// TIA Portal project "tezTia" (V14)

(* hardware
DEVICE "S7-1200 station_1"  S7-1200 Station
   slot 0: "Rack_0"  Rack  V1.0
   slot 1: "PLC_1"  CPU 1215C AC/DC/Rly  6ES7 215-1BG31-0XB0  V3.0
*)

// ===== PLC "PLC_1"  CPU 1215C AC/DC/Rly =====

VAR_GLOBAL   // PLC tag table "Default tag table"
   "start" AT %I0.0 : Bool;
   "stop" AT %I0.1 : Bool;
   "renk sensörü" AT %IW64 : Word;
   "kamera" AT %QW80 : Word;
   "motor" AT %Q0.0 : Bool;
   "motor_1" AT %Q0.1 : Bool;
   "motor_2" AT %Q0.2 : Bool;
   "motor_3" AT %Q0.3 : Bool;
   "motor_4" AT %Q0.4 : Bool;
   "kırmızı" AT %M40.0 : Bool;
   "yeşil" AT %M40.1 : Bool;
   "mavi" AT %M40.2 : Bool;
   "bozuk" AT %M40.3 : Bool;
   "motor_3 geri" AT %Q0.6 : Bool;
END_VAR

DATA_BLOCK "çark çevir_DB"   // DB6
{ S7_Optimized_Access := 'TRUE' }
VERSION : 0.1
// stored: InstanceOfName çark çevir
"çark çevir"
BEGIN
END_DATA_BLOCK

DATA_BLOCK "şekil algıla_DB"   // DB7
{ S7_Optimized_Access := 'TRUE' }
VERSION : 0.1
// stored: InstanceOfName şekil algıla
"şekil algıla"
BEGIN
END_DATA_BLOCK

DATA_BLOCK "reset_DB"   // DB9
{ S7_Optimized_Access := 'TRUE' }
VERSION : 0.1
// stored: InstanceOfName reset
"reset"
BEGIN
END_DATA_BLOCK

// folder: System blocks/Program resources

DATA_BLOCK "IEC_Timer_0_DB"   // DB1
{ S7_Optimized_Access := 'TRUE' }
AUTHOR : Simatic
FAMILY : IEC
NAME : IEC_TMR
VERSION : 1.0
// stored: InstanceOfName IEC_TIMER
"IEC_TIMER"
BEGIN
END_DATA_BLOCK

DATA_BLOCK "IEC_Timer_0_DB_1"   // DB2
{ S7_Optimized_Access := 'TRUE' }
AUTHOR : Simatic
FAMILY : IEC
NAME : IEC_TMR
VERSION : 1.0
// stored: InstanceOfName IEC_TIMER
"IEC_TIMER"
BEGIN
END_DATA_BLOCK

DATA_BLOCK "IEC_Timer_0_DB_2"   // DB3
{ S7_Optimized_Access := 'TRUE' }
AUTHOR : Simatic
FAMILY : IEC
NAME : IEC_TMR
VERSION : 1.0
// stored: InstanceOfName IEC_TIMER
"IEC_TIMER"
BEGIN
END_DATA_BLOCK

DATA_BLOCK "IEC_Timer_0_DB_3"   // DB4
{ S7_Optimized_Access := 'TRUE' }
AUTHOR : Simatic
FAMILY : IEC
NAME : IEC_TMR
VERSION : 1.0
// stored: InstanceOfName IEC_TIMER
"IEC_TIMER"
BEGIN
END_DATA_BLOCK

DATA_BLOCK "IEC_Timer_0_DB_4"   // DB5
{ S7_Optimized_Access := 'TRUE' }
AUTHOR : Simatic
FAMILY : IEC
NAME : IEC_TMR
VERSION : 1.0
// stored: InstanceOfName IEC_TIMER
"IEC_TIMER"
BEGIN
END_DATA_BLOCK

DATA_BLOCK "IEC_Timer_0_DB_5"   // DB8
{ S7_Optimized_Access := 'TRUE' }
AUTHOR : Simatic
FAMILY : IEC
NAME : IEC_TMR
VERSION : 1.0
// stored: InstanceOfName IEC_TIMER
"IEC_TIMER"
BEGIN
END_DATA_BLOCK

// folder: (top level)

FUNCTION_BLOCK "çark çevir"   // FB1, LAD
{ S7_Optimized_Access := 'TRUE' }
VERSION : 0.1
BEGIN

REGION Network 1
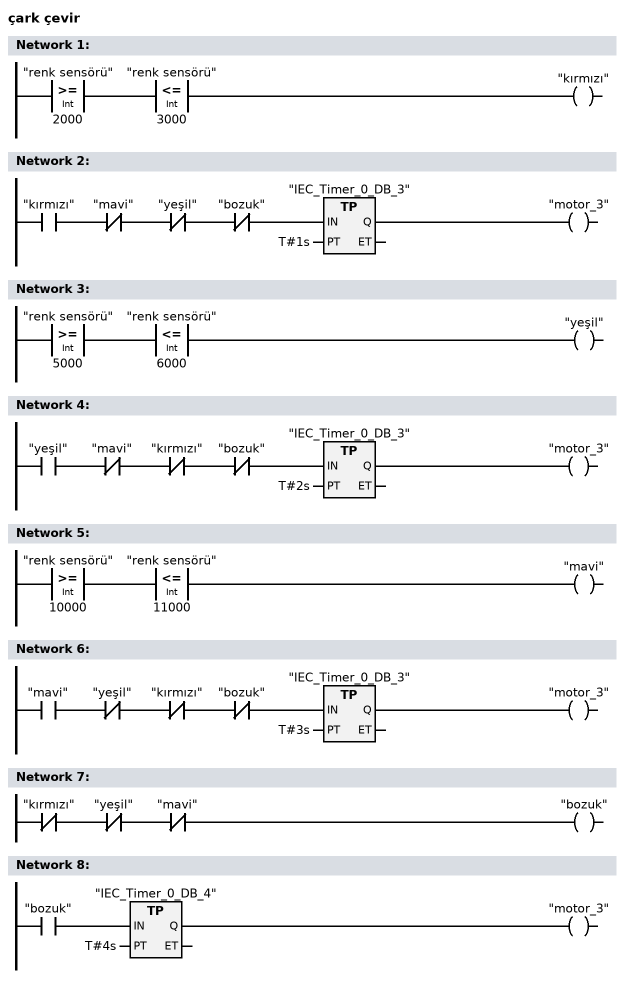
   RUNG wire#powerrail
      { S7_Templates := "SrcType := Int" } GE_Contact(in1 := "renk sensörü", in2 := 2000)
      { S7_Templates := "SrcType := Int" } LE_Contact(in1 := "renk sensörü", in2 := 3000)
      Coil( "kırmızı" )
   END_RUNG
   // the same network as SCL:
   "kırmızı" := ("renk sensörü" >= 2000) AND ("renk sensörü" <= 3000);
END_REGION

REGION Network 2
   "IEC_Timer_0_DB_3".TP(IN := "kırmızı" AND NOT "mavi" AND NOT "yeşil" AND NOT "bozuk", PT := T#1s);
   "motor_3" := "IEC_Timer_0_DB_3".Q;
END_REGION

REGION Network 3
   RUNG wire#powerrail
      { S7_Templates := "SrcType := Int" } GE_Contact(in1 := "renk sensörü", in2 := 5000)
      { S7_Templates := "SrcType := Int" } LE_Contact(in1 := "renk sensörü", in2 := 6000)
      Coil( "yeşil" )
   END_RUNG
   // the same network as SCL:
   "yeşil" := ("renk sensörü" >= 5000) AND ("renk sensörü" <= 6000);
END_REGION

REGION Network 4
   "IEC_Timer_0_DB_3".TP(IN := "yeşil" AND NOT "mavi" AND NOT "kırmızı" AND NOT "bozuk", PT := T#2s);
   "motor_3" := "IEC_Timer_0_DB_3".Q;
END_REGION

REGION Network 5
   RUNG wire#powerrail
      { S7_Templates := "SrcType := Int" } GE_Contact(in1 := "renk sensörü", in2 := 10000)
      { S7_Templates := "SrcType := Int" } LE_Contact(in1 := "renk sensörü", in2 := 11000)
      Coil( "mavi" )
   END_RUNG
   // the same network as SCL:
   "mavi" := ("renk sensörü" >= 10000) AND ("renk sensörü" <= 11000);
END_REGION

REGION Network 6
   "IEC_Timer_0_DB_3".TP(IN := "mavi" AND NOT "yeşil" AND NOT "kırmızı" AND NOT "bozuk", PT := T#3s);
   "motor_3" := "IEC_Timer_0_DB_3".Q;
END_REGION

REGION Network 7
   RUNG wire#powerrail
      I_Contact( "kırmızı" )
      I_Contact( "yeşil" )
      I_Contact( "mavi" )
      Coil( "bozuk" )
   END_RUNG
   // the same network as SCL:
   "bozuk" := NOT "kırmızı" AND NOT "yeşil" AND NOT "mavi";
END_REGION

REGION Network 8
   "IEC_Timer_0_DB_4".TP(IN := "bozuk", PT := T#4s);
   "motor_3" := "IEC_Timer_0_DB_4".Q;
END_REGION
END_FUNCTION_BLOCK

FUNCTION_BLOCK "şekil algıla"   // FB2, LAD
{ S7_Optimized_Access := 'TRUE' }
VERSION : 0.1
BEGIN
END_FUNCTION_BLOCK

FUNCTION_BLOCK "reset"   // FB3, LAD
{ S7_Optimized_Access := 'TRUE' }
VERSION : 0.1
BEGIN

REGION Network 1
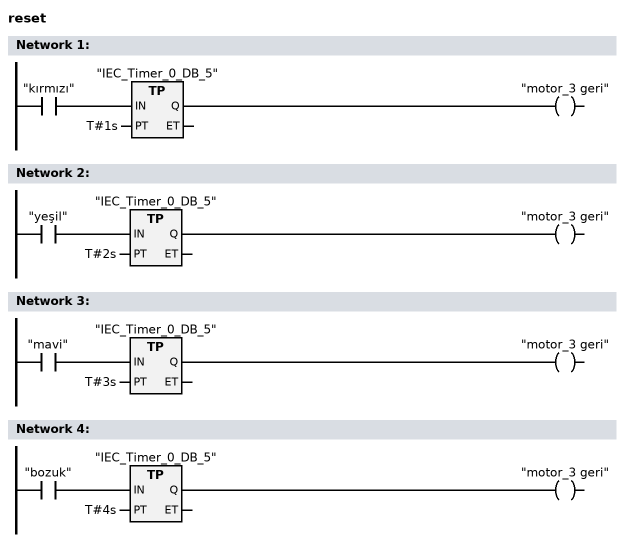
   "IEC_Timer_0_DB_5".TP(IN := "kırmızı", PT := T#1s);
   "motor_3 geri" := "IEC_Timer_0_DB_5".Q;
END_REGION

REGION Network 2
   "IEC_Timer_0_DB_5".TP(IN := "yeşil", PT := T#2s);
   "motor_3 geri" := "IEC_Timer_0_DB_5".Q;
END_REGION

REGION Network 3
   "IEC_Timer_0_DB_5".TP(IN := "mavi", PT := T#3s);
   "motor_3 geri" := "IEC_Timer_0_DB_5".Q;
END_REGION

REGION Network 4
   "IEC_Timer_0_DB_5".TP(IN := "bozuk", PT := T#4s);
   "motor_3 geri" := "IEC_Timer_0_DB_5".Q;
END_REGION
END_FUNCTION_BLOCK

ORGANIZATION_BLOCK "Main"   // OB1, LAD, ProgramCycle
TITLE = "Main Program Sweep (Cycle)"
{ S7_Optimized_Access := 'TRUE' }
VERSION : 0.1
BEGIN

REGION Network 1
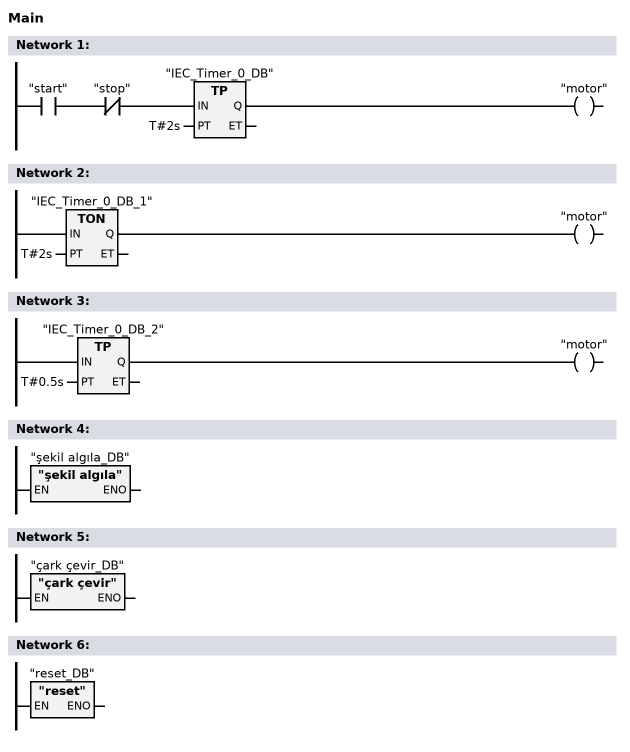
   "IEC_Timer_0_DB".TP(IN := "start" AND NOT "stop", PT := T#2s);
   "motor" := "IEC_Timer_0_DB".Q;
END_REGION

REGION Network 2
   "IEC_Timer_0_DB_1".TON(IN := TRUE, PT := T#2s);
   "motor" := "IEC_Timer_0_DB_1".Q;
END_REGION

REGION Network 3
   "IEC_Timer_0_DB_2".TP(IN := TRUE, PT := T#0.5s);
   "motor" := "IEC_Timer_0_DB_2".Q;
END_REGION

REGION Network 4
   RUNG wire#powerrail
      "şekil algıla_DB"()
   END_RUNG
   // the same network as SCL:
   "şekil algıla_DB"();   // "şekil algıla"
END_REGION

REGION Network 5
   RUNG wire#powerrail
      "çark çevir_DB"()
   END_RUNG
   // the same network as SCL:
   "çark çevir_DB"();   // "çark çevir"
END_REGION

REGION Network 6
   RUNG wire#powerrail
      "reset_DB"()
   END_RUNG
   // the same network as SCL:
   "reset_DB"();   // "reset"
END_REGION
END_ORGANIZATION_BLOCK